PROGRAM MAIN
VAR
	bToggleFlashing : BOOL;
	nCounter: INT;
	bGaugeOn: BOOL;
	
	GaugeTimer: TON;
	GaugeTrig: R_TRIG;
	bGaugeTimerOn: BOOL;
	GaugeCounter: INT;
	
	fbGetLicenses : FB_GetLicensesEx;
	
	iWriteIntHere : INT;
	
END_VAR

nCounter := nCounter +1;

fbGetLicenses.bExecute := true;

IF bGaugeOn THEN
	GaugeTimer(IN:= bGaugeTimerOn, PT:=T#1S , Q=> , ET=> );
	IF GaugeTimer.Q THEN
		bGaugeTimerOn := FALSE;
		GaugeTrig(CLK:= bGaugeOn, Q=> );
		IF GaugeTrig.Q THEN
			GaugeCounter := GaugeCounter + 1;
			bGaugeOn := FALSE;
		END_IF
	END_IF
END_IF

END_PROGRAM

(* stored: Version 1.1.0.1, ProductVersion 3.1.4024.10
   POU MAIN: Id {9dc12211-0425-4f01-97b8-bf7de7386f2f}, SpecialFunc None *)
